(*The tank with opened lid and have a motor for mix, a cylinder for out material*)
FUNCTION_BLOCK FB_Mixer0
VAR
	poCylinderOut : FB_DigitalOutput;
	fbMotorContactor : FB_Contactor1FB_ThermalRelay;
END_VAR

METHOD Mix : BOOL
VAR_INPUT
END_VAR
fbMotorContactor.MR_PowerON();
END_METHOD

METHOD OutMaterial : BOOL
VAR_INPUT
END_VAR
poCylinderOut.Out := true;
END_METHOD

PROPERTY Ref_MotorContactor : REFERENCE TO FB_Contactor1FB_ThermalRelay
GET
Ref_MotorContactor ref= fbMotorContactor;
END_GET
END_PROPERTY

PROPERTY Ref_poCylinderOut : reference to FB_DigitalOutput
GET
Ref_poCylinderOut ref= poCylinderOut;
END_GET
END_PROPERTY

METHOD StopAll : BOOL
VAR_INPUT
END_VAR
StopMix();
StopOutMaterial();
END_METHOD

METHOD StopMix : BOOL
VAR_INPUT
END_VAR
fbMotorContactor.MR_PowerOFF();
END_METHOD

METHOD StopOutMaterial : BOOL
VAR_INPUT
END_VAR
poCylinderOut.Out := false;
END_METHOD

END_FUNCTION_BLOCK

(* stored: Version 1.1.0.1, ProductVersion 3.1.4024.12
   POU FB_Mixer0: Id {b1c4791e-c423-4619-9a92-2d2afdb9cda8}, SpecialFunc None
   Method Mix: Id {e2e02bd9-8fb2-45f0-be31-bd0235cd3989}
   Method OutMaterial: Id {c138c301-8efe-490a-9d86-15f8b54562bc}
   Property Ref_MotorContactor: Id {e9105539-f80b-4827-bb89-f29a8633092f}
   Get Get: Id {2dac6ecd-d27a-429c-b68e-50886cc6dcdb}
   Property Ref_poCylinderOut: Id {29861518-d4a7-4854-bd11-6e5ce0c53288}
   Get Get: Id {827340e2-8f12-4736-9a21-bc71d3cf7333}
   Method StopAll: Id {3d740fe2-2c16-4acd-9e3f-243afaded1b8}
   Method StopMix: Id {9d2b99c9-8201-447e-b61d-8a3a7b0c6f0d}
   Method StopOutMaterial: Id {c1ac88a0-2c74-404a-ba44-65f7eaee8d4e} *)
